Staubli VAL3: loadmaster6.pgx

program loadmaster6(string x_sMasterFile6 (dimensions=1))
begin
  if master:libLoad(x_sMasterFile6)<0
    popUpMsg("nO ok")
  endIf
  frmaster[6].trsf=master:tTool.trsf
  //取个数
  nsize[6]=size(master:ptRoutingPath)
  //存个数
  resize(pdemo6,1,nsize[6])
  //保存程序
  master:libSave()
end
